# EPICS autosave request: support/dac128V-2-6/dac128VApp/Db/DAC_positions.req
# Copy of VME_DAC_positions.req to go along with DAC.db
$(P)$(DAC)_1.VAL
$(P)$(DAC)_2.VAL
$(P)$(DAC)_3.VAL
$(P)$(DAC)_4.VAL
$(P)$(DAC)_5.VAL
$(P)$(DAC)_6.VAL
$(P)$(DAC)_7.VAL
$(P)$(DAC)_8.VAL
